{attribute 'enable_dynamic_creation'}
INTERFACE I_Future EXTENDS __System.IQueryInterface

METHOD abort : BOOL // Return TRUE if finish.
VAR_INPUT
END_VAR
END_METHOD

METHOD error_reset : BOOL
VAR_INPUT
END_VAR
END_METHOD

METHOD execute : BOOL // Return TRUE if finish.
VAR_INPUT
END_VAR
END_METHOD

PROPERTY executor : I_Job
GET
END_GET
SET
END_SET
END_PROPERTY

PROPERTY future_name : STRING // Name of future.
GET
END_GET
SET
END_SET
END_PROPERTY

METHOD init : BOOL // Return TRUE if finish.
VAR_INPUT
END_VAR
END_METHOD

PROPERTY nErrorID : HRESULT // Set result code when finished any method. 0 should be set when normal case.
GET
END_GET
END_PROPERTY

PROPERTY persistent_future : BOOL
GET
END_GET
SET
END_SET
END_PROPERTY

METHOD quit : BOOL // Return TRUE if finish.
VAR_INPUT
END_VAR
END_METHOD

PROPERTY state : E_FutureExecutionState // Execution state of this future.
GET
END_GET
SET
END_SET
END_PROPERTY

END_INTERFACE

(* stored: Version 1.1.0.1, ProductVersion 3.1.4026.17
   Itf I_Future: Id {882bc581-e126-40c6-885e-c12ccc2f0bb9}
   Method abort: Id {527ff0b5-6fbb-4ad6-b3f1-4a79b5e73d86}
   Method error_reset: Id {a9eb976f-3758-4671-96e5-921c7b463a22}
   Method execute: Id {4a0b4721-18ea-4776-928a-5b24c49dda75}
   Property executor: Id {1ffce432-14a7-4918-9f9c-90ae1bb1d90d}
   Get Get: Id {a1986d22-3041-4060-aadc-fc03953d80fb}
   Set Set: Id {cb8b03d6-1988-4e67-b1fe-27b0d43d581d}
   Property future_name: Id {89ef3158-3550-438a-bee3-821a3cca9058}
   Get Get: Id {d6d11718-73bb-4401-91ac-a3e6b656d939}
   Set Set: Id {1b08d5ef-7e1e-4062-a60e-52a0fb1809f4}
   Method init: Id {d56cdce8-543b-417d-80a1-0c782146e5ce}
   Property nErrorID: Id {091e3808-1f21-4039-8bcc-e07988c843df}
   Get Get: Id {3dfc56f5-414c-4e9f-8318-d6a9044e8070}
   Property persistent_future: Id {31178402-da73-4433-b646-5ce9b39fb92c}
   Get Get: Id {3f93484e-26d1-43a7-8e1c-b71a9d011e8a}
   Set Set: Id {76333ad6-86fb-44d3-8bba-0f2650e01274}
   Method quit: Id {12e3433d-9567-4756-bdca-54fc6f4c2614}
   Property state: Id {b673a454-4761-427b-8ab4-14bd1622c60c}
   Get Get: Id {4b1cfb02-a56c-4f6f-980b-64cbecfe2458}
   Set Set: Id {6d81734e-97aa-4d5c-8baf-2d15120c0679} *)
